TYPE sMqttIn :
STRUCT
	sJOB: sJOB;
	sCmd: sCmd;
	boCharging1Connected : BOOL;
	boCharging2Connected : BOOL;
	boNewJob : BOOL;
	END_STRUCT
END_TYPE

(* stored: Version 1.1.0.1, ProductVersion 3.1.4026.13
   DUT sMqttIn: Id {6f2d20af-fcea-4dfd-b27f-99d0e103bd70} *)
